FUNCTION_BLOCK MOTORS_CONSUMPTION (* Peroidic event generator *)
  (* Standard: 61499-1 Annex A; Description: Copyright (c) 2017 fortiss GmbH This program and the accompanying materials are made available under the terms of the Eclipse Public License 2.0 which is available at https://www.eclipse.org/legal/epl-2.0/ SPDX-License-Identifier: EPL-2.0 *)
  (* Version 1.0, 2017-09-21, Alois Zoitl, fortiss GmbH, initial API and implementation and/or initial documentation *)
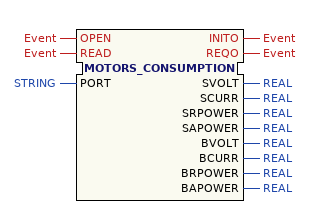
  EVENT_INPUT
    OPEN;
    READ;
  END_EVENT
  EVENT_OUTPUT
    INITO;
    REQO;
  END_EVENT
  VAR_INPUT
    PORT : STRING;
  END_VAR
  VAR_OUTPUT
    SVOLT : REAL;
    SCURR : REAL;
    SRPOWER : REAL;
    SAPOWER : REAL;
    BVOLT : REAL;
    BCURR : REAL;
    BRPOWER : REAL;
    BAPOWER : REAL;
  END_VAR
END_FUNCTION_BLOCK
